// TIA Portal V20 export
TYPE "zp_CITI_Parameters"
// stored: Namespace CITI_Logic
   STRUCT
      Map_ID : SInt;   // Map Number for Reference in Data
      MachineType : SInt;   // Set the Machine Type According to the Following - (1=Machine_Assembly; 2=Filter_Coolant; 3=CMM)
      Rtd_CycTime : DInt := 0;   // Rated Cycle Time in mSec
      Flt_Det_Dly : Int := 0;   // Fault Detect Delay Time in mSec
      DTT_IN : Int;   // Delay Transfer Time IN
      DTT_OUT : Int;   // Delay Transfer Time OUT
      CycTime_DataDly : DInt := 0;   // Cycletime Data Delay Time in mSec
      CycleTime_Data_Dwll : DInt := 0;   // Cycletime Data Dwell Time in mSec
      Parts_Per_Cyc : Int := 0;   // Parts Per Cycle
      RetryCnt : Int := 0;   // Process Retry Count
      FlasherRate : Int := 0;   // Flasher Rate msec
   END_STRUCT;
END_TYPE
